TYPE ST_ITC_GSR :
(**************************************************************************************
 * 	Application		:	BoxControl Framework
 *	Revision		:	$Revision: 404529 $
 *	Revision date	:	$Date: 2018-04-23 08:21:38 +0200 (Mo., 23 Apr 2018) $
 *	Last changed by	:	$Author: b7bolm $
 *	URL				:	$URL: http://almscdc.swisslog.com/repo/SWPD/Development/BoxControlFramework/20_Release/trunk/01_Software/BCF/BCF/JumpStart/20_Product/10_App/11_Com/10_Lib/10_Conv/11_ITC/01_DUTs/ST_ITC_GSR.TcDUT $
 *
 *	Purpose			:	GCR Structure
 *
 * ------------------------------------------------------------------------------------
 *	Copyright Swisslog [IP AG], Switzerland. All rights reserved.
 * 
 * ------------------------------------------------------------------------------------
 *	
 * 	Revision History: 
 *
 * 	VERSION			DATE			INITIALS			DESCRIPTION
 *	0.1				01.01.2001		swl					Example
 *
 **************************************************************************************)
STRUCT
	GroupName			: STRING(Conveyor.POSITION_STRINGLENGTH); // 12 Digit SIS Group Name MM-GGG-0000-000 
	eMode				: E_PositionMode; // Mode
	eState				: E_PositionState; // State
	eErrorState			: E_ErrorState; // Error State
	eErrorCode			: E_ErrorConv; // Return Code
	eErrorType			: E_ErrorType; // Error Type
	ErrorInformation	: STRING(System.ERROR_PARAM_STRINGLENGTH); // 5 Chars Error Information
	Variable			: DINT; // Variable
	eReturnCode			: E_ErrorConv; // Return code
END_STRUCT
END_TYPE

(* stored: Version 1.1.0.1, ProductVersion 3.1.4022.12
   DUT ST_ITC_GSR: Id {fe56e7ac-9495-4e01-980d-4861188d0a01} *)
